// TIA Portal V20 export
DATA_BLOCK "SiCom"   // DB48
{ S7_Optimized_Access := 'TRUE' }
// stored: AutoNumber false, MemoryReserve 100
   VAR
      Ack : Bool;   // reset faults general
      LampTest : Struct   // lamp test
         SettingMode : Bool;   // setting mode
         LaserOn : Bool;   // laser on
         XrayOn : Bool;   // xray on
      END_STRUCT;
      Blinker : Bool;   // blinker
      Flash : Bool;   // flash
      SafetyTest : Bool;   // safety test
      AreaLaserOn : Bool;   // area laser on
      AreaAdjustmentOn : Bool;   // area adjustment on
      AreaXrayOn : Bool;   // area X-Ray on
      ResetSafetyDevice : Bool;   // reset safety devices
   END_VAR
BEGIN
END_DATA_BLOCK
